FUNCTION_BLOCK FB_ObjectBase_V2 IMPLEMENTS IBasicElement
VAR_INPUT
    Execute    :BOOL;   // True : This prog will start.
    Abort      :BOOL;   // True : This prog will be abort.
    Reset      :BOOL;   // True : This prog will be reset.
    ObjectName :STRING; // Set this fb name(About it's action)
END_VAR

VAR_OUTPUT
    Busy    :BOOL;        // True : This prog is running.
    Done    :BOOL;        // True : Command has been executed.
    Aborted :BOOL;        // True : This prog is aborted.
    Error   :BOOL;        // True : This prog has an error.
    ErrorID :UINT;       // Output ErrorID
    Status  :STRING; // Output this prog status by string(255bytes)
	UniqueErrorCode :STRING;	
END_VAR

VAR
    eState :E_MethodStatus_Basic;
	uiExecutingStep : UDINT; // This var is used to been controll STATE_EXECUTING process.
	uiResettingStep : UDINT;
	uiAbortingStep : UDINT;
	_Executed :BOOL; // Executing process completed.
	_Error : BOOL; // FB has an error.
	_ResetCompleted : BOOL; // FB resetting completed.
	_AbortCompleted : BOOL; // FB aborting completed.
END_VAR

A00_BasicUnits();
A10_StateControl();

ACTION A00_BasicUnits:

END_ACTION

ACTION A10_StateControl:
CASE eState OF
	STATE_DORMANT:
		M_STATE_DORMANT();
	STATE_EXECUTING:
		M_STATE_EXECUTING();
	STATE_ABORTING:
		M_STATE_ABORTING();
	STATE_ABORTED:
		M_STATE_ABORTED();
	STATE_DONE:
		M_STATE_DONE();
	STATE_ERROR:
		M_STATE_ERROR();
	STATE_RESETTING:
		M_STATE_RESETTING();
END_CASE
END_ACTION

METHOD GetModelState
VAR_OUTPUT
    xDone    :BOOL;
    xBusy    :BOOL;
    xError   :BOOL;
    xAborted :BOOL;
    iErrorID :UDINT;	
	UniqueErrorCode : STRING;
END_VAR
xDone    := Done;
xBusy    := Busy;
xError   := Error;
xAborted := Abort;
iErrorID := ErrorID;
UniqueErrorCode := THIS^.UniqueErrorCode;
END_METHOD

METHOD GetName : STRING
GetName := ObjectName;
END_METHOD

METHOD M_RefLinks
VAR_INPUT
END_VAR
END_METHOD

METHOD  M_STATE_ABORTED
VAR_INPUT
END_VAR
;
END_METHOD

METHOD  M_STATE_ABORTING
VAR_INPUT
END_VAR
;
END_METHOD

METHOD  M_STATE_DONE
VAR_INPUT
END_VAR
;
END_METHOD

METHOD  M_STATE_DORMANT
VAR_INPUT
END_VAR
;
END_METHOD

METHOD  M_STATE_ERROR
VAR_INPUT
END_VAR
;
END_METHOD

METHOD  M_STATE_EXECUTING
VAR_INPUT
END_VAR
;
END_METHOD

METHOD  M_STATE_RESETTING
VAR_INPUT
END_VAR
;
END_METHOD

END_FUNCTION_BLOCK

(* stored: Version 1.1.0.1, ProductVersion 3.1.4024.13
   POU FB_ObjectBase_V2: Id {9a229dbf-569c-4d2e-b613-f9255a5a7b3c}, SpecialFunc None
   Folder STATE: Id {f29bc40c-f94c-4d00-9112-4fc5f7479e02}
   Action A00_BasicUnits: Id {e7beb950-0ff4-452f-ad21-f987036a0354}
   Action A10_StateControl: Id {1cecd68d-19c8-433e-8666-d30d4916d754}
   Method GetModelState: Id {02e18dc0-d842-4f77-87d5-8645879337b1}
   Method GetName: Id {fcad8b4f-3c87-4c54-a85b-c334a7010435}
   Method M_RefLinks: Id {b1e0f55a-91c7-406a-8907-94fe5bddb966}
   Method M_STATE_ABORTED: Id {04eff820-bbb8-4cc6-a29d-96d8b5a052f3}
   Method M_STATE_ABORTING: Id {32b36f9e-9b49-4ded-aa25-f6b1e7b7b786}
   Method M_STATE_DONE: Id {c00cc89d-031d-49e6-8d51-62dedf9ce7d2}
   Method M_STATE_DORMANT: Id {3816a803-4d71-4329-95b9-f217fd3a6a05}
   Method M_STATE_ERROR: Id {1edd602d-fb03-4bfc-a73f-f32d0970a717}
   Method M_STATE_EXECUTING: Id {29ca477a-9cf8-41da-a9a9-6580a546527a}
   Method M_STATE_RESETTING: Id {cca28a45-fe94-4a4d-885c-859aa5e0107c} *)
